TYPE ST_KomunikatorKolejka :
STRUCT
	stKomunikat					: ST_KomunikatorKomunikat;
	bWysylanie					: BOOL;
	bPotwierdzenie				: BOOL;
	itfNadawca					: ITF_KomunikatorNadawca;
	itfOdbiorca					: ITF_KomunikatorOdbiorca;
	
END_STRUCT
END_TYPE

(* stored: Version 1.1.0.1
   DUT ST_KomunikatorKolejka: Id {f3df0a22-2d82-062c-18b5-7c2b5a82b67e} *)
